// TIA Portal V17 export
// export: Created 2024-08-09T12:53:18.9330927Z, ExportSetting WithDefaults, DisplayName Totally Integrated Automation Portal, DisplayVersion V17 Update 7, DisplayName TIA Portal Openness, DisplayVersion V17 Update 7, DisplayName TIA Portal Version Control Interface, DisplayVersion V17, DisplayName STEP 7 Professional, DisplayVersion V17 Update 7, DisplayName STEP 7 Safety, DisplayVersion V17 Update 6, DisplayName WinCC Professional, DisplayVersion V17 Update 7
TYPE "S_Derout_Exp"
// stored: IsFailsafeCompliant false
   STRUCT
      CommunDos : "S_Dosage_Commun";
      Pt_Zs : "S_Suivi_Dosage";
      Dial_Def { S7_SetPoint := 'True'} : "S_DIALOG_DEF";
      Fg_Derout : Bool;
      Fg_Valid_Ctrl_Incomp_Cir_Cel : Bool;
      Pt_Cel { S7_SetPoint := 'True'} : "S_Cellule";
      Lst_Taches_Att_Deb_Mel { ExternalAccessible := 'False'; ExternalVisible := 'False'; ExternalWritable := 'False'} : Array[0.."T_MAX_AMONTAVAL"] of "S_TacheNiv";
      Lst_Taches_Att_Fin_Mel { S7_SetPoint := 'True'} : Array[0.."T_MAX_AMONTAVAL"] of "S_TacheNiv";
      Lst_Taches_Maj_Cel_Suiv { S7_SetPoint := 'True'} : Array[0.."T_MAX_AMONTAVAL"] of "S_TacheNiv";
   END_STRUCT;
END_TYPE
